PROGRAM MAIN
VAR
END_VAR

END_PROGRAM

(* stored: Version 1.1.0.1
   POU MAIN: Id {72e74c75-036f-41d0-9197-90f78f7ff78b} *)
